// TwinCAT 3 PLC project MAS418_PLC
// ProgramVersion: 3.1.4023.0
// libraries:
//   Tc2_Standard, * (Beckhoff Automation GmbH)
//   Tc2_System, * (Beckhoff Automation GmbH)
//   Tc3_Module, * (Beckhoff Automation GmbH)
//   VisuDialogs, * (System)
//   VisuSymbols,3.5.10.0,System
// project tree:
//   DUTs/ Sensies.TcDUT
//   / GlobalTextList.TcGTLO, PlcTask.TcTTO, Visualization Manager.TcVMO (not stored)
//   GVLs/ DB.TcGVL, G_Task2.TcGVL, ST_Timer.TcDUT
//   POUs/ DegToRad.TcPOU, MAIN.TcPOU
//   VISUs/ Visualization.TcVIS
// real-time tasks:
//   TASK PlcTask: cycle T#10ms, priority 20, ADS port 350

CONFIGURATION MAS418_PLC
    RESOURCE PLC ON TwinCAT3
        TASK PlcTask(INTERVAL := T#10ms, PRIORITY := 20);
        PROGRAM MAIN WITH PlcTask : MAIN;
    END_RESOURCE
END_CONFIGURATION

// ---- DUTs/Sensies.TcDUT
{attribute 'qualified_only'}
{attribute 'strict'}
TYPE Sensies :
(
	Sick := 0,
	Pilz := 1,
	Parker := 2,
	Bosh := 3
)USINT;
END_TYPE

// ---- GVLs/ST_Timer.TcDUT
TYPE ST_Timer :
STRUCT
	StartTimer : BOOL := TRUE;
	TimeToPass : TIME;
	CurrentTime : TIME;
	IsFinished : BOOL := FALSE;
END_STRUCT
END_TYPE

// ---- GVLs/DB.TcGVL
VAR_GLOBAL
	dtVariable : DATE_AND_TIME := DT#2023-02-08-15:31:19;
	pToString : POINTER TO STRING;
	var2 : TIME := T#5S;
	var2Ref: REFERENCE TO TIME;
	var3 : ARRAY[1..4] OF DATE := [D#2023-02-7, D#2023-02-8, D#2023-02-9, D#2023-02-10];
	
	Sensor1 : Sensies := Sensies.Parker;
	
	TimeToPass : TIME := T#10S;
	Timmie : TON := (PT := TimeToPass);
	StartTimer : BOOL := FALSE;
	CurrentTimmie : TIME;
	IsFinished : BOOL;
	
END_VAR

// ---- GVLs/G_Task2.TcGVL
VAR_GLOBAL
	Timer2 : ST_Timer := (TimeToPass:= T#5S);
	TimerTof : TOF := (PT := Timer2.TimeToPass, Q := Timer2.IsFinished);
	Motor1 : LREAL := 180;
	Motor2 : LREAL;

END_VAR

// ---- POUs/MAIN.TcPOU
PROGRAM MAIN
VAR
	bEnable : BOOL;
	bStart : BOOL;
	
END_VAR

bEnable := bStart;

pToString := ADR(dtVariable);
var2Ref REF= var2;

Timmie(IN := StartTimer);

CurrentTimmie := Timmie.ET;

TimerTof(IN := Timer2.StartTimer);
Timer2.CurrentTime := Timer2.CurrentTime;

DegToRad(Degval := Motor1,
		Radval => Motor2);

END_PROGRAM

// ---- POUs/DegToRad.TcPOU
FUNCTION DegToRad : LREAL
VAR_INPUT
	Degval : LREAL;
END_VAR
VAR_OUTPUT
	Radval : LREAL := (DegVal*(PI/180));
END_VAR

END_FUNCTION

// ---- GlobalTextList.TcGTLO
TEXTLIST GlobalTextList
  243 = '%f'
  27 = '%i'
  955 = '%s'
  517 = 'BOOL'
  745 = 'DataTypeTesting'
  596 = 'INT'
  124 = 'Lamp'
  73 = 'REAL'
  426 = 'STRING'
  40 = 'UINT'
END_TEXTLIST

// ---- VISUs/Visualization.TcVIS
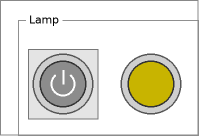
VISUALIZATION Visualization  // 199x136
    GroupBox (18,12 181x124), "Lamp"
        PowerSwitch (10,37 70x70), variable: MAIN.bStart, behaviour: TOGGLE, style: Switch-PowerSwitch-Gray
        Lamp1 (98,37 70x70), variable: MAIN.bEnable, style: Lamp-Lamp1-Yellow
END_VISUALIZATION
